PROGRAM blink
VAR
	start AT %IX0.0 : bool;
	coil : bool;
	stop AT %IX0.1 : bool;
	led AT %QX0.0 : bool;
	TON0 : TON;
	TOF0 : TOF;
	TON1 : TON;
	TOF1 : TOF;
END_VAR
  VAR  (* added by the conversion: wires and edge detectors of the diagram *)
    _TON11_ET : ANY;
    _TON11_OUT : BOOL;
    _TOF12_ET : ANY;
    _TOF12_OUT : BOOL;
  END_VAR

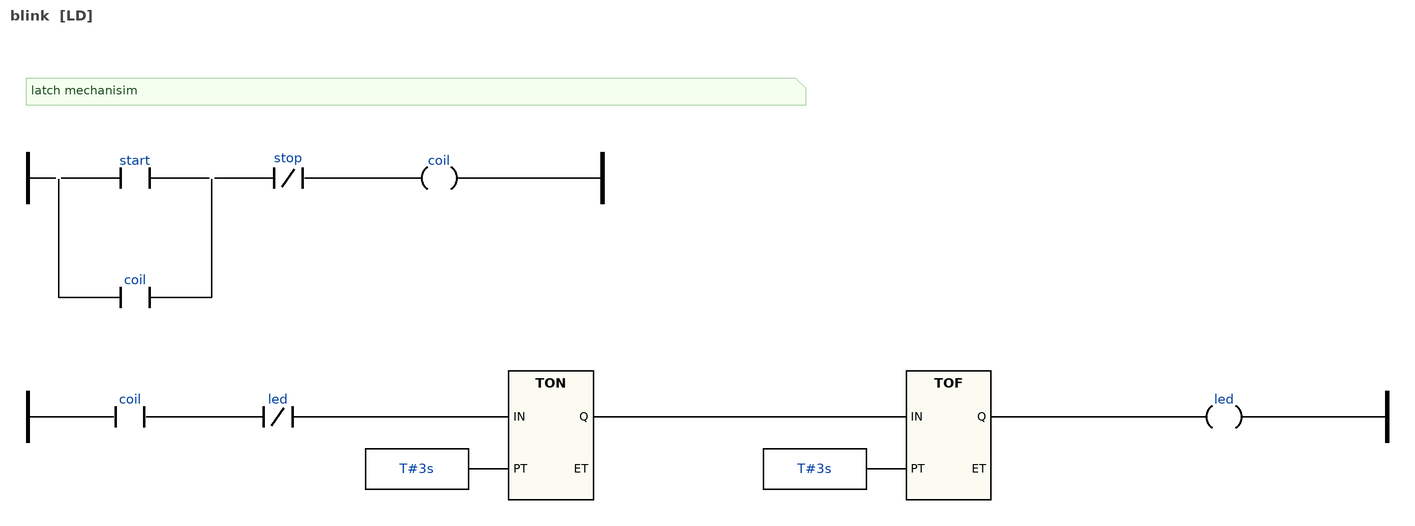
(* LD diagram, written out as Structured Text *)
(* latch mechanisim *)
coil := (start OR coil) AND NOT stop;
_TON11_OUT := TON(IN := coil AND NOT led, PT := T#3s, ET => _TON11_ET);
_TOF12_OUT := TOF(IN := _TON11_OUT, PT := T#3s, ET => _TOF12_ET);
led := _TOF12_OUT;
END_PROGRAM
